TYPE ST_IO2_InputPLC :
STRUCT
	bRawInput			: BOOL;
	bRawRTrigger			: BOOL;
	bRawFTrigger			: BOOL;
	bStateInput			: BOOL;
	bStateRTrigger			: BOOL;
	bStateFTrigger			: BOOL;
END_STRUCT
END_TYPE

(* stored: Version 1.1.0.1, ProductVersion 3.1.4024.15
   DUT ST_IO2_InputPLC: Id {2ef7afa2-8da0-48aa-a4be-6b1d81ae200d} *)
